Fanuc KAREL source: NC0002.compact.KL

PROGRAM NC0002
%STACKSIZE=65535
%PRIORITY=65535
%NOLOCKGROUP
ROUTINE R FROM NC0002
ROUTINE R
VAR
S1 : INTEGER
BEGIN
S1=1
IF (S1=1) THEN
S1=(S1 + 1)
ELSE
S1=(S1 + 2)
ENDIF
END R
BEGIN
R
END NC0002
